// TwinCAT 3 PLC project PlcProj
// ProgramVersion: 3.1.4024.12
// libraries:
//   Tc2_BABasic, * (Beckhoff Automation GmbH)
//   Tc2_Drive, * (Beckhoff Automation GmbH)
//   Tc2_MC2, * (Beckhoff Automation GmbH)
//   Tc2_MC2_Drive, * (Beckhoff Automation GmbH)
//   Tc2_NcKinematicTransformation, * (Beckhoff Automation GmbH)
//   Tc2_PlcInterpolation, * (Beckhoff Automation GmbH)
//   Tc2_Standard, * (Beckhoff Automation GmbH)
//   Tc2_System, * (Beckhoff Automation GmbH)
//   Tc2_Utilities, * (Beckhoff Automation GmbH)
//   Tc3_McCoordinatedMotion, * (Beckhoff Automation GmbH)
//   Tc3_Module, * (Beckhoff Automation GmbH)
// project tree:
//   FBs/ FB_CalculateLinkageArm.TcPOU, FB_EnableAxes.TcPOU, FB_ResetCoordinateAxes.TcPOU
//   GVLs/ GVL.TcGVL
//   / PlcTask.TcTTO
//   POUs/ MAIN.TcPOU
// real-time tasks:
//   TASK PlcTask: cycle T#10ms, priority 20, ADS port 350
//   TASK Job Task: cycle default, priority 32
// motion (NC):
//   TASK NC-Task 1 SAF: cycle T#2ms, priority 4, ADS port 501
//   TASK NC-Task 1 SVB: cycle T#10ms, priority 8, ADS port 511
//   AXIS M1 (ACS) Degrees (id 1)
//     PositionAreaControl: Enable=false, Range=0
//     OtherSettings: AllowMotionCmdToSlave=true
//     encoder EncType=1
//     drive DrvType=5
//       Analog: TorqueSetpointScale=10, ScaleFactorActTorque=0.1
//       TimeComp: TaskDelayCycles=1
//     controller CtrType=1
//       CtrPara: PriorControlFactor=1
//         PosDiffControl: Enable=false, Range=0
//         Observer: BandWidth=20
//   AXIS M2 (ACS) Degrees (id 2)
//     PositionAreaControl: Enable=false, Range=0
//     OtherSettings: AllowMotionCmdToSlave=true
//     encoder EncType=1
//     drive DrvType=5
//       Analog: TorqueSetpointScale=10, ScaleFactorActTorque=0.1
//       TimeComp: TaskDelayCycles=1
//     controller CtrType=1
//       CtrPara: PriorControlFactor=1
//         PosDiffControl: Enable=false, Range=0
//         Observer: BandWidth=20
//   AXIS M3 (ACS) mm (id 3)
//     PositionAreaControl: Enable=false, Range=0
//     OtherSettings: AllowMotionCmdToSlave=true
//     encoder EncType=1
//     drive DrvType=5
//       Analog: TorqueSetpointScale=10, ScaleFactorActTorque=0.1
//       TimeComp: TaskDelayCycles=1
//     controller CtrType=1
//       CtrPara: PriorControlFactor=1
//         PosDiffControl: Enable=false, Range=0
//         Observer: BandWidth=20
//   AXIS M4 (ACS) Degrees (id 4)
//     PositionAreaControl: Enable=false, Range=0
//     OtherSettings: AllowMotionCmdToSlave=true
//     encoder EncType=1
//     drive DrvType=5
//       Analog: TorqueSetpointScale=10, ScaleFactorActTorque=0.1
//       TimeComp: TaskDelayCycles=1
//     controller CtrType=1
//       CtrPara: PriorControlFactor=1
//         PosDiffControl: Enable=false, Range=0
//         Observer: BandWidth=20
//   AXIS X (MCS) (id 5)
//     OtherSettings: AllowMotionCmdToSlave=true
//     encoder EncType=1
//     drive DrvType=5
//       Analog: TorqueSetpointScale=10, ScaleFactorActTorque=0.1
//       TimeComp: TaskDelayCycles=1
//     controller CtrType=1
//       CtrPara: PriorControlFactor=1
//         Observer: BandWidth=20
//   AXIS Y (MCS) (id 6)
//     OtherSettings: AllowMotionCmdToSlave=true
//     encoder EncType=1
//     drive DrvType=5
//       Analog: TorqueSetpointScale=10, ScaleFactorActTorque=0.1
//       TimeComp: TaskDelayCycles=1
//     controller CtrType=1
//       CtrPara: PriorControlFactor=1
//         Observer: BandWidth=20
//   AXIS Z (MCS) (id 7)
//     OtherSettings: AllowMotionCmdToSlave=true
//     encoder EncType=1
//     drive DrvType=5
//       Analog: TorqueSetpointScale=10, ScaleFactorActTorque=0.1
//       TimeComp: TaskDelayCycles=1
//     controller CtrType=1
//       CtrPara: PriorControlFactor=1
//         Observer: BandWidth=20
//   AXIS C (MCS) (id 8)
//     OtherSettings: AllowMotionCmdToSlave=true
//     encoder EncType=1
//     drive DrvType=5
//       Analog: TorqueSetpointScale=10, ScaleFactorActTorque=0.1
//       TimeComp: TaskDelayCycles=1
//     controller CtrType=1
//       CtrPara: PriorControlFactor=1
//         Observer: BandWidth=20
// variable links:
//   PlcProj/PlcProj Instance <-> NC-Task 1 SAF/Axes/C (MCS)
//     PlcTask Inputs/MAIN.io_C.NcToPlc <-> Outputs/ToPlc
//     PlcTask Outputs/MAIN.io_C.PlcToNc <-> Inputs/FromPlc
//   PlcProj/PlcProj Instance <-> NC-Task 1 SAF/Axes/M1 (ACS) Degrees
//     PlcTask Inputs/MAIN.io_M1.NcToPlc <-> Outputs/ToPlc
//     PlcTask Outputs/MAIN.io_M1.PlcToNc <-> Inputs/FromPlc
//   PlcProj/PlcProj Instance <-> NC-Task 1 SAF/Axes/M2 (ACS) Degrees
//     PlcTask Inputs/MAIN.io_M2.NcToPlc <-> Outputs/ToPlc
//     PlcTask Outputs/MAIN.io_M2.PlcToNc <-> Inputs/FromPlc
//   PlcProj/PlcProj Instance <-> NC-Task 1 SAF/Axes/M3 (ACS) mm
//     PlcTask Inputs/MAIN.io_M3.NcToPlc <-> Outputs/ToPlc
//     PlcTask Outputs/MAIN.io_M3.PlcToNc <-> Inputs/FromPlc
//   PlcProj/PlcProj Instance <-> NC-Task 1 SAF/Axes/M4 (ACS) Degrees
//     PlcTask Inputs/MAIN.io_M4.NcToPlc <-> Outputs/ToPlc
//     PlcTask Outputs/MAIN.io_M4.PlcToNc <-> Inputs/FromPlc
//   PlcProj/PlcProj Instance <-> NC-Task 1 SAF/Axes/X (MCS)
//     PlcTask Inputs/MAIN.io_X.NcToPlc <-> Outputs/ToPlc
//     PlcTask Outputs/MAIN.io_X.PlcToNc <-> Inputs/FromPlc
//   PlcProj/PlcProj Instance <-> NC-Task 1 SAF/Axes/Y (MCS)
//     PlcTask Inputs/MAIN.io_Y.NcToPlc <-> Outputs/ToPlc
//     PlcTask Outputs/MAIN.io_Y.PlcToNc <-> Inputs/FromPlc
//   PlcProj/PlcProj Instance <-> NC-Task 1 SAF/Axes/Z (MCS)
//     PlcTask Inputs/MAIN.io_Z.NcToPlc <-> Outputs/ToPlc
//     PlcTask Outputs/MAIN.io_Z.PlcToNc <-> Inputs/FromPlc
//   PlcProj/PlcProj Instance <-> NC-Task 1 SAF/Kinematics Channel
//     PlcTask Inputs/MAIN.in_stKinToPlc <-> Outputs/ToPlc
//     PlcTask Outputs/MAIN.out_stPlcToKin <-> Inputs/FromPlc
//   PlcProj/PlcProj Instance <-> NC-Task 1 SAF/Objects/Motion Group
//     PlcTask Inputs/GVL.stGroupRef.NcToPlc <-> Group Outputs/ToPLC
//     PlcTask Outputs/GVL.stGroupRef.PlcToNc <-> Group Inputs/FromPLC

CONFIGURATION PlcProj
    RESOURCE PLC ON TwinCAT3
        TASK PlcTask(INTERVAL := T#10ms, PRIORITY := 20);
        PROGRAM MAIN WITH PlcTask : MAIN;
    END_RESOURCE
END_CONFIGURATION

// ---- GVLs/GVL.TcGVL
{attribute 'qualified_only'}
VAR_GLOBAL
	
	stGroupRef : AXES_GROUP_REF;
	{attribute 'TcInitSymbol'}  oidConveyorBelt : MC_COORD_REF;

	
END_VAR

// ---- POUs/MAIN.TcPOU
PROGRAM MAIN
VAR
	
	inner_arm : FB_CalculateLinkageArm;
	outer_arm : FB_CalculateLinkageArm;
	
	io_X:	AXIS_REF;
	io_Y:	AXIS_REF;
	io_Z:	AXIS_REF;
	io_C:	AXIS_REF;	
	io_M1:	AXIS_REF;
	io_M2:	AXIS_REF;
	io_M3:	AXIS_REF;
	io_M4:	AXIS_REF;	

	fbAddAxisXtoGrp : MC_AddAxisToGroup;
	fbAddAxisYtoGrp : MC_AddAxisToGroup;
	fbAddAxisZtoGrp : MC_AddAxisToGroup;	
	fbAddAxisCtoGrp : MC_AddAxisToGroup;	
	
//	Kinematic Functions / Structures / Vars
	bkinConfigGrp				: BOOL;
	bkinCartesianMode			: BOOL := TRUE; //When bCartesianMode is TRUE, movement in the MCS (Cartesian) axes will be transformed into the ACS (Joint) axes. The ACS axes cannot be moved directly.
	bkinResetGrp					: BOOL;
	in_stKinToPlc	AT %I*		: NcToPlc_NciChannel_Ref;
	out_stPlcToKin	AT %Q*		: PLCTONC_NCICHANNEL_REF;
	stAxesConfig				: ST_KinAxes;
	fbCalcTrafo					: FB_KinCalcTrafo;
	metaIn						: U_KinMetaInfo;
	metaOut						: U_KinMetaInfo;
	fbKinConfigGrp				: FB_KinConfigGroup;  //Configures ACS and MCS axes to the kinematic transformation group
	fbKinResetGrp				: FB_KinResetGroup;  //Resets the kinematic transformation group
	oidTrafo		AT %I*		: OTCID;
	kinStatus 					: E_KinStatus;
	
	bDeltaKinEnable : BOOL;
	bDeltaKinReady : BOOL;
	bDeltaKinActive : BOOL;
	bDeltaKinInactive : BOOL;
	nDeltaKinState : INT;
	
	bKinGrpEnable : BOOL;
	bKinGrpReady : BOOL;
	bKinGrpError : BOOL;
	bKinGrpReset : BOOL;
	bNciEnable : BOOL;
	bKinResetDone : BOOL;
	bNciReadytToEnable : BOOL;
	bEnableAxes : BOOL;
	bAllAxesReady : BOOL;
	fbKinDelay : TON;
	fbEnableAxes : FB_EnableAxes;
	bAxisFault : BOOL;
	fbResetCoordinateAxes : FB_ResetCoordinateAxes;
	fbJogX : MC_Jog;
	fbJogY : MC_Jog;
	fbJogZ : MC_Jog;
	fbMoveX : MC_MoveRelative;
	bMoveX : BOOL;
	nDistanceX : INT;
	nDistanceY : INT;
	nDistanceZ : INT;
	bMoveY : BOOL;
	bMoveZ : BOOL;
	fbMoveY : MC_MoveRelative;
	fbMoveZ : MC_MoveRelative;
	bAxesNotMoving : BOOL;
	bJogXpos : BOOL;
	bJogXneg : BOOL;
	nMoveState	: WORD;
	
	bMotionGrpEnable : BOOL;	// Enable the Motion Group
	bMotionGrpBuild : BOOL;		// Add Axes To Motion Group
	bMotionGrpStop : BOOL;
	bMotionGrpStart : BOOL;
	bMotionGrpPrep : BOOL;
	bMotionGrpOvr : BOOL;
	
	fbMgSetOverride : MC_GroupSetOverride;
	fbMgEnable : MC_GroupEnable;
	fbMoveLinPrep : MC_MoveLinearAbsolutePreparation;
	fbMoveCircPrep : MC_MoveCircularAbsolutePreparation;
	fbMgMovePath : MC_MovePath;
	fbMgStop 	: MC_GroupStop;
	fbMgReadStatus : MC_GroupReadStatus;
	
	// hmi
	
	nDisplayZ : LREAL;
	nPkgZ   : LREAL;
	nScaleZ : LREAL;
	nDisplayX : LREAL;
	nDisplayY : LREAL;
	
	
	// copied from sample proj
	
	buffer					: ARRAY[1..4096] OF BYTE;
	path					: MC_PATH_DATA_REF(ADR(buffer), SIZEOF(buffer));
	
	aTargetPos				: ARRAY[1..4] OF MC_LREAL;
	aTransitionParam		: ARRAY[1..2] OF MC_LREAL;
	aAuxPoint                               : ARRAY[1..3] OF MC_LREAL;
	fVelFactor				: LREAL := 1.0;
	bMovePrepError : BOOL;
	bBarPicked : BOOL;
	bAddNewBar : BOOL;
	fbAddNewBar : TON;
	bBarPlaced : BOOL;
	nBarDisplayX : LREAL;
	nBarDisplayY : LREAL;
	nBarDisplayZ : LREAL;
	bNewPath	: BOOL;
	bBarInPlace  : BOOL;
	nTestBarX : LREAL;
	nTestBarY : LREAL;
	nTestBarZ : LREAL;
		nScaledBarX : LREAL;
	nScaledBarY : LREAL;
	nScaledBarZ : LREAL;
	
	
	fbTrackConveyor : MC_TrackConveyorBelt;
	MasterRefPos : MC_LREAL;
	InitialObjectPos : ARRAY [1..4] OF MC_LREAL;
	bStartTracking : BOOL;
	fbStartConveyor : MC_MoveVelocity;
	fbStopConveyor : MC_Stop;
	bStartConveyor : BOOL;
	bStopGroup : BOOL;
	lrYpos: MC_LREAL;
	fbSetM1Pos : MC_SetPosition;
	fbSetM2Pos : MC_SetPosition;
	fbSetM4Pos : MC_SetPosition;
	bSetPos : BOOL;
	
	nTrackX: LREAL;
END_VAR


// action calls
	Main.cartesian_ops();
	Main.kinematic_ops();
	Main.motion_group();

// calculations for hmi display of the scara linkages
	inner_arm(
		x0:= 375, 
		y0:= 375, 
		theta:= io_M1.NcToPlc.ActPos, 
		L:= 190, 
		x1=> , 
		y1=> );
	
	outer_arm(
		x0:= inner_arm.x1, 
		y0:= inner_arm.y1, 
		theta:= io_M2.NcToPlc.ActPos, 
		L:= 190, 
		x1=> , 
		y1=> );

// Axis Ref Read Status
	io_X.ReadStatus();
	io_Y.ReadStatus();
	io_Z.ReadStatus();
	io_C.ReadStatus();	
	io_M1.ReadStatus();
	io_M2.ReadStatus();
	io_M3.ReadStatus();
	io_M4.ReadStatus();	

// check for motor movement
	bAxesNotMoving := io_M1.Status.NotMoving AND io_M2.Status.NotMoving AND io_M3.Status.NotMoving AND io_M4.Status.NotMoving;
	
// read axes id's from cylic interface so they can mapped later to the kinematic group
	stAxesConfig.nAxisIdsAcs[1]	:= io_M1.NcToPlc.AxisId;
	stAxesConfig.nAxisIdsAcs[2]	:= io_M2.NcToPlc.AxisId;
	stAxesConfig.nAxisIdsAcs[3]	:= io_M3.NcToPlc.AxisId;
	stAxesConfig.nAxisIdsAcs[4]	:= io_M4.NcToPlc.AxisId;	
	stAxesConfig.nAxisIdsMcs[1]	:= io_X.NcToPlc.AxisId;
	stAxesConfig.nAxisIdsMcs[2]	:= io_Y.NcToPlc.AxisId;
	stAxesConfig.nAxisIdsMcs[3]	:= io_Z.NcToPlc.AxisId;
	stAxesConfig.nAxisIdsMcs[4]	:= io_C.NcToPlc.AxisId;	
	

	fbMgMovePath(
		AxesGroup:= GVL.stGroupRef , 
		PathData:= path , 
		Execute:= bMotionGrpStart
	);
	
	fbMgStop(
		AxesGroup := GVL.stGroupRef,
		Execute	:= bStopGroup
		);
	
			
CASE nMoveState OF
	
1:	//	init

		nMoveState	:= 4;
		
4:	// set up path data for the pick position

		Main.prep_pick_path();
		//Main.prep_start_path();
		
		IF path.FilledRows > 0 THEN
			nMoveState	:= 5;
		END_IF
		
5:	// move to the pick psoition

		bMotionGrpStart := TRUE;

		IF fbMgMovePath.Done THEN
			bMotionGrpStart := FALSE;
			nMoveState := 100;
		END_IF

10:	// set up path data for the place position

		Main.prep_place_path();
		//Main.prep_finish_path();
		
		IF path.FilledRows > 0 THEN
			nMoveState	:= 15;
		END_IF
		
15:	// move to the place position

		bMotionGrpStart := TRUE;

		IF fbMgMovePath.Done THEN
			bMotionGrpStart := FALSE;
			nMoveState := 1;
		END_IF

100: // stopping...

		bStopGroup := TRUE;
		
		IF fbMgStop.Done THEN
			bStopGroup := FALSE;
			nMoveState	:= 10;
		END_IF		

END_CASE

ACTION cartesian_ops:
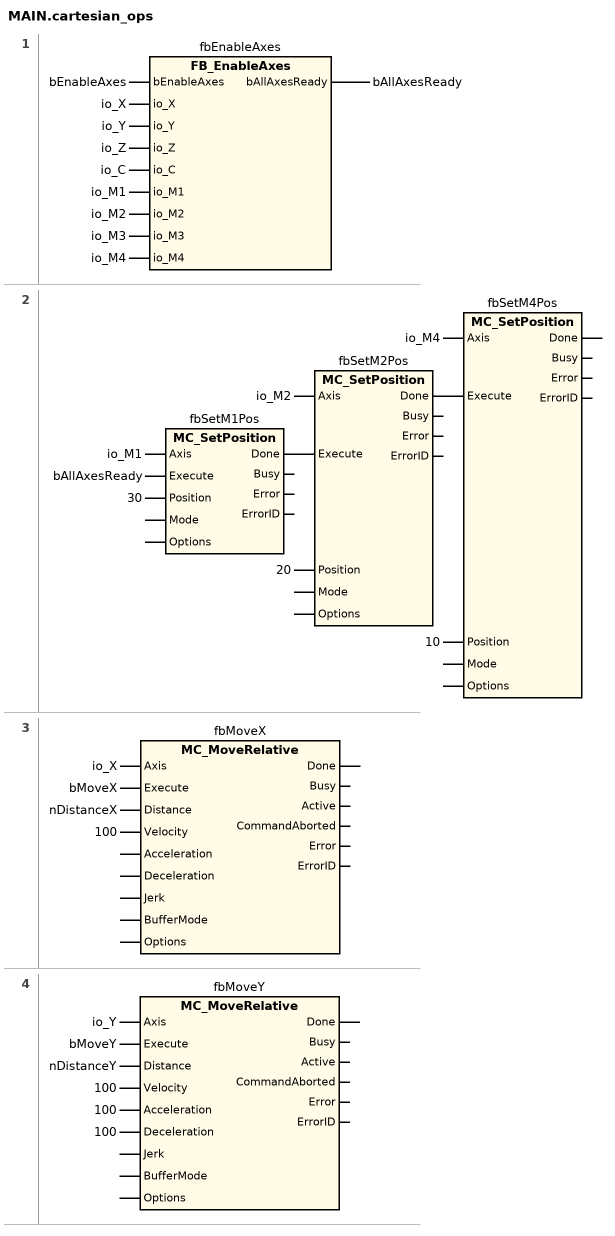
// NETWORK 1
fbEnableAxes(
    bEnableAxes := bEnableAxes,
    io_X := io_X,
    io_Y := io_Y,
    io_Z := io_Z,
    io_C := io_C,
    io_M1 := io_M1,
    io_M2 := io_M2,
    io_M3 := io_M3,
    io_M4 := io_M4); // FB_EnableAxes
bAllAxesReady := fbEnableAxes.bAllAxesReady;

// NETWORK 2
fbSetM1Pos(Axis := io_M1, Execute := bAllAxesReady, Position := 30); // MC_SetPosition
fbSetM2Pos(Axis := io_M2, Execute := fbSetM1Pos.Done, Position := 20); // MC_SetPosition
fbSetM4Pos(Axis := io_M4, Execute := fbSetM2Pos.Done, Position := 10); // MC_SetPosition

// NETWORK 3
fbMoveX(Axis := io_X, Execute := bMoveX, Distance := nDistanceX, Velocity := 100); // MC_MoveRelative

// NETWORK 4
fbMoveY(
    Axis := io_Y,
    Execute := bMoveY,
    Distance := nDistanceY,
    Velocity := 100,
    Acceleration := 100,
    Deceleration := 100); // MC_MoveRelative

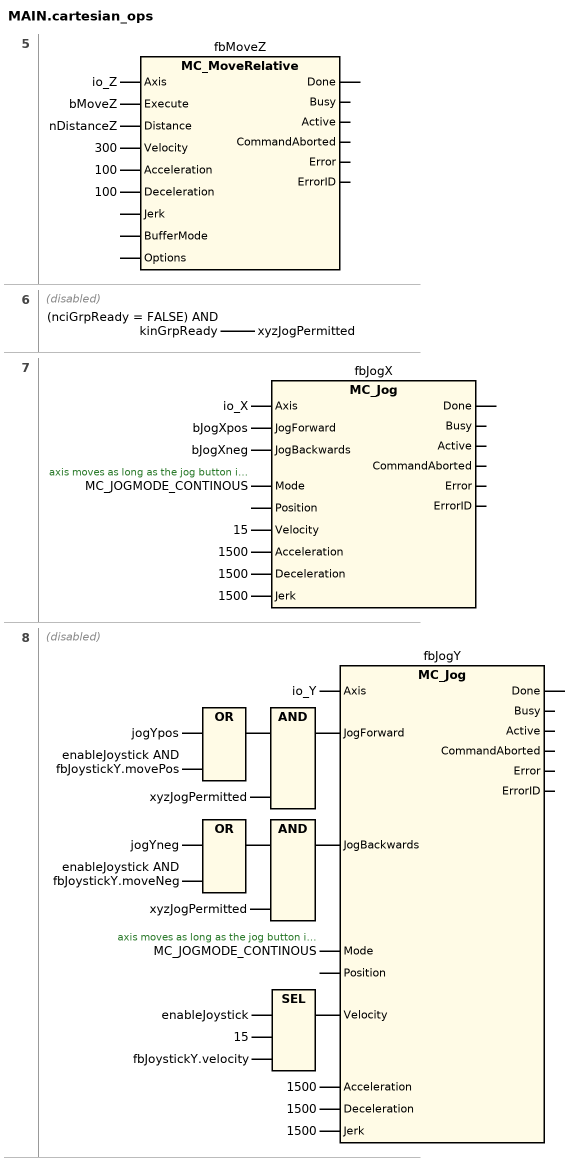
// NETWORK 5
fbMoveZ(
    Axis := io_Z,
    Execute := bMoveZ,
    Distance := nDistanceZ,
    Velocity := 300,
    Acceleration := 100,
    Deceleration := 100); // MC_MoveRelative

// NETWORK 6 (disabled)
// xyzJogPermitted := (nciGrpReady = FALSE) AND kinGrpReady;

// NETWORK 7
//   MC_JOGMODE_CONTINOUS: axis moves as long as the jog button is pressed using parameterized dynamics
fbJogX(
    Axis := io_X,
    JogForward := bJogXpos,
    JogBackwards := bJogXneg,
    Mode := MC_JOGMODE_CONTINOUS,
    Velocity := 15,
    Acceleration := 1500,
    Deceleration := 1500,
    Jerk := 1500); // MC_Jog

// NETWORK 8 (disabled)
//   MC_JOGMODE_CONTINOUS: axis moves as long as the jog button is pressed using parameterized dynamics
// fbJogY(
//     Axis := io_Y,
//     JogForward := (jogYpos OR (enableJoystick AND fbJoystickY.movePos)) AND xyzJogPermitted,
//     JogBackwards := (jogYneg OR (enableJoystick AND fbJoystickY.moveNeg)) AND xyzJogPermitted,
//     Mode := MC_JOGMODE_CONTINOUS,
//     Velocity := SEL(enableJoystick, 15, fbJoystickY.velocity),
//     Acceleration := 1500,
//     Deceleration := 1500,
//     Jerk := 1500); // MC_Jog

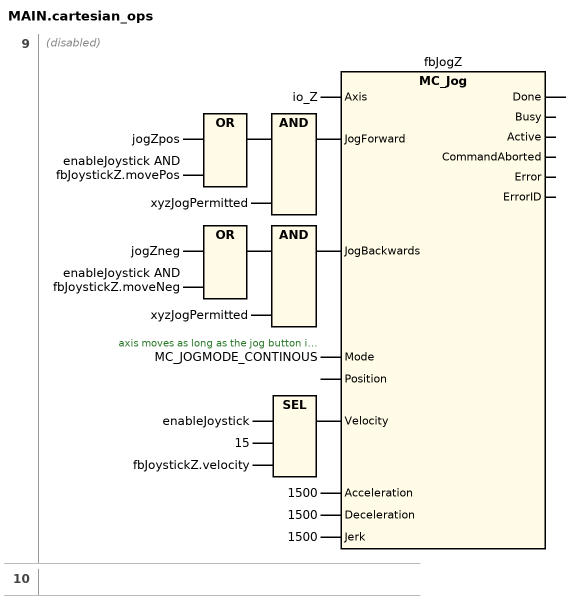
// NETWORK 9 (disabled)
//   MC_JOGMODE_CONTINOUS: axis moves as long as the jog button is pressed using parameterized dynamics
// fbJogZ(
//     Axis := io_Z,
//     JogForward := (jogZpos OR (enableJoystick AND fbJoystickZ.movePos)) AND xyzJogPermitted,
//     JogBackwards := (jogZneg OR (enableJoystick AND fbJoystickZ.moveNeg)) AND xyzJogPermitted,
//     Mode := MC_JOGMODE_CONTINOUS,
//     Velocity := SEL(enableJoystick, 15, fbJoystickZ.velocity),
//     Acceleration := 1500,
//     Deceleration := 1500,
//     Jerk := 1500); // MC_Jog

// NETWORK 10
END_ACTION

ACTION kinematic_ops:
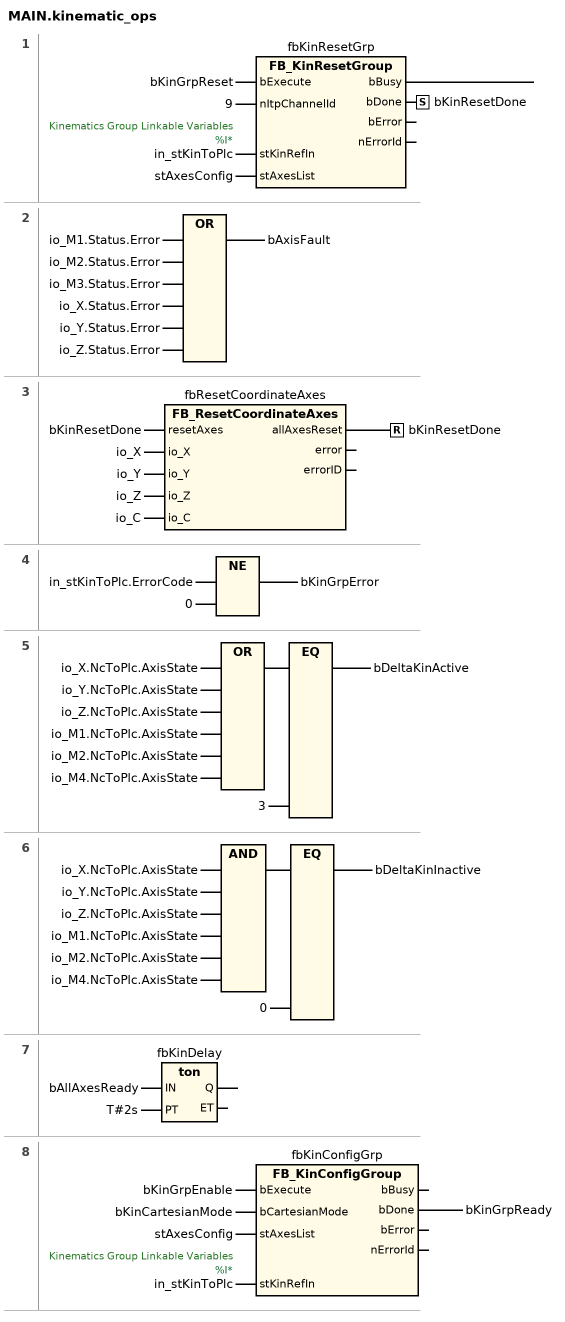
// NETWORK 1
//   fbKinResetGrp: Resets the kinematic transformation group
//   in_stKinToPlc: Kinematics Group Linkable Variables | AT %I*
fbKinResetGrp(
    bExecute := bKinGrpReset,
    nItpChannelId := 9,
    stKinRefIn := in_stKinToPlc,
    stAxesList := stAxesConfig); // FB_KinResetGroup
bKinResetDone S= fbKinResetGrp.bDone;

// NETWORK 2
bAxisFault := io_M1.Status.Error OR io_M2.Status.Error OR io_M3.Status.Error OR io_X.Status.Error OR io_Y.Status.Error OR io_Z.Status.Error;

// NETWORK 3
fbResetCoordinateAxes(resetAxes := bKinResetDone, io_X := io_X, io_Y := io_Y, io_Z := io_Z, io_C := io_C); // FB_ResetCoordinateAxes
bKinResetDone R= fbResetCoordinateAxes.allAxesReset;

// NETWORK 4
bKinGrpError := in_stKinToPlc.ErrorCode <> 0;

// NETWORK 5
bDeltaKinActive := (io_X.NcToPlc.AxisState OR io_Y.NcToPlc.AxisState OR io_Z.NcToPlc.AxisState OR io_M1.NcToPlc.AxisState OR io_M2.NcToPlc.AxisState OR io_M4.NcToPlc.AxisState) = 3;

// NETWORK 6
bDeltaKinInactive := (io_X.NcToPlc.AxisState AND io_Y.NcToPlc.AxisState AND io_Z.NcToPlc.AxisState AND io_M1.NcToPlc.AxisState AND io_M2.NcToPlc.AxisState AND io_M4.NcToPlc.AxisState) = 0;

// NETWORK 7
fbKinDelay(IN := bAllAxesReady, PT := T#2s); // ton

// NETWORK 8
//   fbKinConfigGrp: Configures ACS and MCS axes to the kinematic transformation group
//   in_stKinToPlc: Kinematics Group Linkable Variables | AT %I*
fbKinConfigGrp(
    bExecute := bKinGrpEnable,
    bCartesianMode := bKinCartesianMode,
    stAxesList := stAxesConfig,
    stKinRefIn := in_stKinToPlc); // FB_KinConfigGroup
bKinGrpReady := fbKinConfigGrp.bDone;

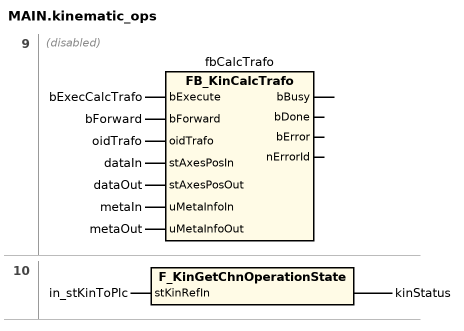
// NETWORK 9 (disabled)
// fbCalcTrafo(
//     bExecute := bExecCalcTrafo,
//     bForward := bForward,
//     oidTrafo := oidTrafo,
//     stAxesPosIn := dataIn,
//     stAxesPosOut := dataOut,
//     uMetaInfoIn := metaIn,
//     uMetaInfoOut := metaOut); // FB_KinCalcTrafo

// NETWORK 10
kinStatus := F_KinGetChnOperationState(stKinRefIn := in_stKinToPlc);
END_ACTION

ACTION kinematic_sm:

(*
		setStartPos[5](Axis:= io_X, 
			Execute:= setZeroPosition,
			Position:= 0);
		setStartPos[6](Axis:= io_Y,
			Execute:= setZeroPosition, 
			Position:= 0);
		setStartPos[7](Axis:= io_Z, 
			Execute:= setZeroPosition,
			Position:= 0);
*)

CASE nDeltaKinState OF 

0: 	nDeltaKinState := 2;

		
2:			// RESET ALL NCI VARIABLES
		//nciRunProgram := FALSE;
		//nciBuildTable := FALSE;
		//nciResetTable := TRUE;
		//nciResetProgram := TRUE;
		nDeltaKinState := 3;
		
3:
		//nciResetProgram := FALSE;
		//nciResetTable := FALSE;
		nDeltaKinState := 4;
		
4:			// RESET ALL KINEMATIC VARIABLES
		IF bKinGrpError THEN
				bKinGrpReset := TRUE;
				nDeltaKinState :=5;
		ELSIF bKinGrpError = FALSE THEN
				nDeltaKinState := 104;
		END_IF
				
5:
		bKinGrpReset := FALSE;
		nDeltaKinState := 4;
		
104:		// RESET ALL KINEMATIC VARIABLES
		IF bAxisFault THEN
				bKinGrpReset := TRUE;
				nDeltaKinState :=105;
		ELSIF bAxisFault = FALSE THEN
				nDeltaKinState := 6;
		END_IF
				
105:
		bKinGrpReset := FALSE;
		nDeltaKinState := 104;

6: 		// IF IN START POSITION - ENABLE AXES
		nDeltaKinState := 7;

7:			// ALL AXES ARE POWERED
		IF bAllAxesReady AND bAxesNotMoving THEN
				nDeltaKinState := 8;
		END_IF
		
8:			// ENABLE KINEMATIC GROUP FUNCTION
		nDeltaKinState := 9;
			
9: 		// DELAY TO ALLOW KINEMATIC GROUP TIME TO PROCESS REQUEST
		IF fbKinDelay.Q AND bKinGrpReady AND bAxesNotMoving THEN
				nDeltaKinState := 10;
		END_IF
	(*	
10:		// ENABLE NCI BUILD GROUP

		nDeltaKinState := 11;

11: 	// WAIT FOR BUILD GROUP DONE AND ADDITIONAL DELAY BEFORE STARTING BUILD TABLE
		IF kinGrpReady  AND  tNciDelay.Q THEN 
				nciBuildTable := TRUE;
				nDeltaKinState := 12;
		ELSIF kinGrpReady = FALSE THEN
				nDeltaKinState := 50;
		END_IF

12: 	// WAIT FOR ROWS TO BE FILLED

		IF fbNciFeedTablePrep.nFilledRows > 0 THEN
				nciBuildTable := FALSE;
				nDeltaKinState:= 13;
		END_IF

13:	// RUN COMMAND WILL START THE NCI FEED TABLE PROGRAM
		IF nciRunCmd  THEN
				nciRunProgram := TRUE; 	
				nDeltaKinState :=14;
		ELSIF nciEnable = FALSE THEN
				nDeltaKinState := 0;
		END_IF
		
14:	
		IF nciFeedingDone THEN
				nciRunProgram := FALSE;
				nDeltaKinState := 15;
		ELSIF nciEnable = FALSE THEN
				nDeltaKinState := 0;
		END_IF

15:	// REACHED END OF FEED TABLE PROGRAM
		IF fbNciTable.bChannelDone THEN
				nDeltaKinState	:= 16;
		ELSIF nciEnable = FALSE THEN
				nDeltaKinState := 0;
		END_IF
		
16:	// IF RUN IS STILL ACTIVE, LOOP BACK THROUGH THE FEED TABLE PROGRAM

		nDeltaKinState := 13;


50: // DECOUPLE KINEMATIC GROUP FROM AXES
		kinCartesianMode := FALSE;
		kinGrpEnable := TRUE;
		
		IF kinStatus = KinStatus_Empty THEN
				kinCartesianMode := TRUE;
				kinGrpEnable := FALSE;
				nDeltaKinState := 4;
		END_IF
	*)			
END_CASE
END_ACTION

ACTION motion_group:
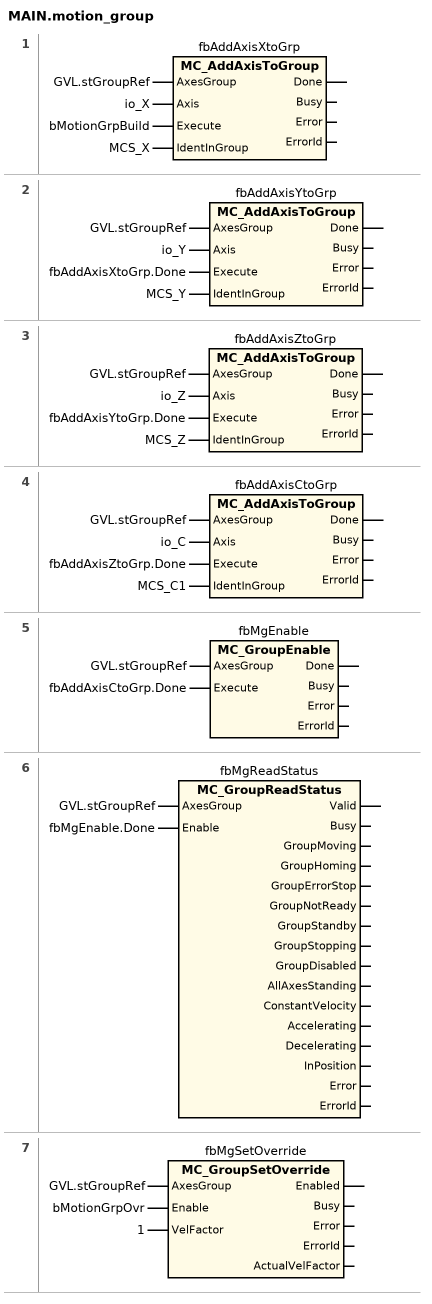
// NETWORK 1
fbAddAxisXtoGrp(AxesGroup := GVL.stGroupRef, Axis := io_X, Execute := bMotionGrpBuild, IdentInGroup := MCS_X); // MC_AddAxisToGroup

// NETWORK 2
fbAddAxisYtoGrp(
    AxesGroup := GVL.stGroupRef,
    Axis := io_Y,
    Execute := fbAddAxisXtoGrp.Done,
    IdentInGroup := MCS_Y); // MC_AddAxisToGroup

// NETWORK 3
fbAddAxisZtoGrp(
    AxesGroup := GVL.stGroupRef,
    Axis := io_Z,
    Execute := fbAddAxisYtoGrp.Done,
    IdentInGroup := MCS_Z); // MC_AddAxisToGroup

// NETWORK 4
fbAddAxisCtoGrp(
    AxesGroup := GVL.stGroupRef,
    Axis := io_C,
    Execute := fbAddAxisZtoGrp.Done,
    IdentInGroup := MCS_C1); // MC_AddAxisToGroup

// NETWORK 5
fbMgEnable(AxesGroup := GVL.stGroupRef, Execute := fbAddAxisCtoGrp.Done); // MC_GroupEnable

// NETWORK 6
fbMgReadStatus(AxesGroup := GVL.stGroupRef, Enable := fbMgEnable.Done); // MC_GroupReadStatus

// NETWORK 7
fbMgSetOverride(AxesGroup := GVL.stGroupRef, Enable := bMotionGrpOvr, VelFactor := 1); // MC_GroupSetOverride
END_ACTION

ACTION prep_finish_path:

path.ClearPath();  //Clear nodes that were in path


// XYZ POSITIONS LIMITS
// X : -760 to +760
// Y : -760 to +760
// Z : 



fbMoveCircPrep.EndPoint                 	:= ADR(aTargetPos);
fbMoveCircPrep.EndPointCount            	:= 4;
fbMoveCircPrep.AuxPoint                 	:= ADR(aTransitionParam);
fbMoveCircPrep.AuxPointCount            	:= 3;
fbMoveCircPrep.CircMode                 	:= mcCircModeCenter;
fbMoveCircPrep.TransitionParameter      	:= ADR(aTransitionParam);
fbMoveCircPrep.TransitionParameterCount 	:= 2;
fbMoveCircPrep.BufferMode               	:= mcBlendingPrevious;
fbMoveCircPrep.TransitionMode           	:= mcTransModeNone;
	
fbMoveLinPrep.Position						:= ADR(aTargetPos); //pointer to position array
fbMoveLinPrep.PositionCount 				:= 4; //number of axes in group
fbMoveLinPrep.TransitionParameter			:= ADR (aTransitionParam); //pointer to transition parameter array
fbMoveLinPrep.TransitionParameterCount		:= 2; //number of transition parameters, has to be set always 2
fbMoveLinPrep.BufferMode					:= mcBlendingPrevious;
fbMoveLinPrep.TransitionMode				:= mcTransModeCornerDistanceAdvanced;

//Set dynamics to default values of the axes
fbMoveLinPrep.Acceleration					:= MC_DEFAULT;
fbMoveLinPrep.Deceleration					:= MC_DEFAULT;
fbMoveLinPrep.Jerk							:= MC_DEFAULT;

bMovePrepError := bMovePrepError OR fbMoveLinPrep.Error;



  	aTargetPos[1]                           := 625;
    aTargetPos[2]                           := 10;
    aTargetPos[3]                           := 0;
    aTransitionParam[1]                     := 0;
    aTransitionParam[2]                     := 0;
    fbMoveLinPrep(PathData:= path, Velocity:= 100, InvokeId:= 10);

    aTargetPos[1]                           := -400;
    aTargetPos[2]                           := -300;
    aTargetPos[3]                           := 0;
    aAuxPoint[1]                            := -357.5;
    aAuxPoint[2]                            := -257.5;
    aAuxPoint[3]                            := 0;
    aTransitionParam[1]                     := 0;
    aTransitionParam[2]                     := 0;
    fbMoveCircPrep(PathData:= path, PathChoice:= mcCircPathchoiceClockwise, Velocity:= 100, InvokeId:= 20);
END_ACTION

ACTION prep_pick_path:
path.ClearPath();  //Clear nodes that were in path


// XYZ POSITIONS LIMITS
// X : -760 to +760
// Y : -760 to +760
// Z : 

//1st node
aTargetPos[1]				:=634;		// X Position
aTargetPos[2]				:= 10;		// Y Position
aTargetPos[3]				:= 0;	// Z Position
aTargetPos[4]				:= 0;	// C Position
aTransitionParam[1]			:= 0; //blending distance on previous segment, no influence here
aTransitionParam[2]			:= 0; //blending distance on this segment, no influence here
fbMoveLinPrep(PathData:= path , Velocity:= 200, InvokeId:= 10);
bMovePrepError := bMovePrepError OR fbMoveLinPrep.Error;

fbMoveLinPrep.Position						:= ADR(aTargetPos); //pointer to position array
fbMoveLinPrep.PositionCount 				:= 4; //number of axes in group
fbMoveLinPrep.TransitionParameter			:= ADR (aTransitionParam); //pointer to transition parameter array
fbMoveLinPrep.TransitionParameterCount		:= 2; //number of transition parameters, has to be set always 2
fbMoveLinPrep.BufferMode					:= mcBlendingPrevious;
fbMoveLinPrep.TransitionMode				:= mcTransModeCornerDistanceAdvanced;
//Set dynamics to default values of the axes
fbMoveLinPrep.Acceleration					:= MC_DEFAULT;
fbMoveLinPrep.Deceleration					:= MC_DEFAULT;
fbMoveLinPrep.Jerk							:= MC_DEFAULT;
END_ACTION

ACTION prep_place_path:
path.ClearPath();  //Clear nodes that were in path

// XYZ POSITIONS LIMITS
// X : -550 to +550
// Y : -550 to +550
// Z : -750 to -950

fbMoveLinPrep.Position						:= ADR(aTargetPos); //pointer to position array
fbMoveLinPrep.PositionCount 				:= 4; //number of axes in group
fbMoveLinPrep.TransitionParameter			:= ADR (aTransitionParam); //pointer to transition parameter array
fbMoveLinPrep.TransitionParameterCount		:= 2; //number of transition parameters, has to be set always 2
fbMoveLinPrep.BufferMode					:= mcBlendingPrevious;
fbMoveLinPrep.TransitionMode				:= mcTransModeCornerDistanceAdvanced;
//Set dynamics to default values of the axes
fbMoveLinPrep.Acceleration					:= MC_DEFAULT;
fbMoveLinPrep.Deceleration					:= MC_DEFAULT;
fbMoveLinPrep.Jerk							:= MC_DEFAULT;
(*
//1st node
aTargetPos[1]				:= -225;		// X Position
aTargetPos[2]				:= 225;		// Y Position
aTargetPos[3]				:= -900;	// Z Position
aTransitionParam[1]			:= 0; //blending distance on previous segment, no influence here
aTransitionParam[2]			:= 0; //blending distance on this segment, no influence here
fbMoveLinPrep(PathData:= path , Velocity:= 2100, InvokeId:= 10);
bMovePrepError := bMovePrepError OR fbMoveLinPrep.Error;

aTargetPos[1]				:= 225;
aTargetPos[2]				:= -225;
aTargetPos[3]				:= -750;
aTransitionParam[1]			:= 50; //blending distance on previous segment (InvokeId=10), defines when to leave line
aTransitionParam[2]			:= 50; //blending distance on this segment, defines latest positionn to be back  on line of InovkeId=20 
fbMoveLinPrep(PathData:= path , Velocity:= 2100, InvokeId:= 20); 
bMovePrepError := bMovePrepError OR fbMoveLinPrep.Error;

aTargetPos[1]				:= 225;
aTargetPos[2]				:= 225;
aTargetPos[3]				:= -950;
aTransitionParam[1]			:= 50; 
aTransitionParam[2]			:= 50;
fbMoveLinPrep(PathData:= path , Velocity:= 2100, InvokeId:= 30);
bMovePrepError := bMovePrepError OR fbMoveLinPrep.Error;

aTargetPos[1]				:= -225;
aTargetPos[2]				:= -225;
aTargetPos[3]				:= -750;
aTransitionParam[1]			:= 50; //blending distance on previous segment, no influence here
aTransitionParam[2]			:= 50; //blending distance on this segment, no influence here
fbMoveLinPrep(PathData:= path , Velocity:= 2100, InvokeId:= 40);
bMovePrepError := bMovePrepError OR fbMoveLinPrep.Error;
*)
aTargetPos[1]				:= -400;
aTargetPos[2]				:= -300;
aTargetPos[3]				:= 0;
aTargetPos[4]				:= 0;
aTransitionParam[1]			:= 50; 
aTransitionParam[2]			:= 50;
fbMoveLinPrep(PathData:= path , Velocity:= 150, InvokeId:= 50);
bMovePrepError := bMovePrepError OR fbMoveLinPrep.Error;
END_ACTION

ACTION prep_start_path:

path.ClearPath();  //Clear nodes that were in path


// XYZ POSITIONS LIMITS
// X : -760 to +760
// Y : -760 to +760
// Z : 



fbMoveCircPrep.EndPoint                 	:= ADR(aTargetPos);
fbMoveCircPrep.EndPointCount            	:= 4;
fbMoveCircPrep.AuxPoint                 	:= ADR(aTransitionParam);
fbMoveCircPrep.AuxPointCount            	:= 3;
fbMoveCircPrep.CircMode                 	:= mcCircModeCenter;
fbMoveCircPrep.TransitionParameter      	:= ADR(aTransitionParam);
fbMoveCircPrep.TransitionParameterCount 	:= 2;
fbMoveCircPrep.BufferMode               	:= mcBlendingPrevious;
fbMoveCircPrep.TransitionMode           	:= mcTransModeNone;
	
fbMoveLinPrep.Position						:= ADR(aTargetPos); //pointer to position array
fbMoveLinPrep.PositionCount 				:= 4; //number of axes in group
fbMoveLinPrep.TransitionParameter			:= ADR (aTransitionParam); //pointer to transition parameter array
fbMoveLinPrep.TransitionParameterCount		:= 2; //number of transition parameters, has to be set always 2
fbMoveLinPrep.BufferMode					:= mcBlendingPrevious;
fbMoveLinPrep.TransitionMode				:= mcTransModeCornerDistanceAdvanced;

//Set dynamics to default values of the axes
fbMoveLinPrep.Acceleration					:= MC_DEFAULT;
fbMoveLinPrep.Deceleration					:= MC_DEFAULT;
fbMoveLinPrep.Jerk							:= MC_DEFAULT;

bMovePrepError := bMovePrepError OR fbMoveLinPrep.Error;



  	aTargetPos[1]                           := -350;
    aTargetPos[2]                           := -300;
    aTargetPos[3]                           := 0;
    aTransitionParam[1]                     := 0;
    aTransitionParam[2]                     := 0;
    fbMoveLinPrep(PathData:= path, Velocity:= 100, InvokeId:= 10);

    aTargetPos[1]                           := 625;
    aTargetPos[2]                           := -10;
    aTargetPos[3]                           := 0;
    aAuxPoint[1]                            := 282.5;
    aAuxPoint[2]                            := -642.5;
    aAuxPoint[3]                            := 0;
    aTransitionParam[1]                     := 0;
    aTransitionParam[2]                     := 0;
    fbMoveCircPrep(PathData:= path, PathChoice:= mcCircPathChoiceCounterClockwise, Velocity:= 100, InvokeId:= 20);
END_ACTION

END_PROGRAM

// ---- FBs/FB_CalculateLinkageArm.TcPOU
FUNCTION_BLOCK FB_CalculateLinkageArm
VAR_INPUT
		x0 : REAL; 			(* Origin x-coordinate *)
        y0 : REAL; 			(* Origin y-coordinate *)
        theta : LREAL ;		(* Angle in degrees *)
        L : REAL ;			(* Length of the line *)

END_VAR

VAR_OUTPUT
	    x1 : REAL;			(* End x-coordinate *)
        y1 : REAL;			(* End y-coordinate *)
END_VAR
VAR
	        theta_rad : REAL;	(* Angle in radians *)
END_VAR

    theta_rad := theta * 3.14159265358979 / 180.0;  

	x1 := x0 + L * COS(theta_rad);
	y1 := y0 + L * SIN(theta_rad);

END_FUNCTION_BLOCK

// ---- FBs/FB_EnableAxes.TcPOU
FUNCTION_BLOCK FB_EnableAxes
VAR_INPUT
	bEnableAxes: BOOL := TRUE;
END_VAR
VAR_OUTPUT
	bAllAxesReady: BOOL := FALSE;
END_VAR
VAR_IN_OUT
	io_X: AXIS_REF;
	io_Y: AXIS_REF;
	io_Z: AXIS_REF;
	io_C: AXIS_REF;
	io_M1: AXIS_REF;
	io_M2: AXIS_REF;
	io_M3: AXIS_REF;
	io_M4 : AXIS_REF;
END_VAR
VAR
	fOverride: LREAL := 100.0;
	fbPowerX: MC_Power;
	fbPowerY: MC_Power;
	fbPowerZ: MC_Power;
	fbPowerC: MC_Power;	
	fbPowerM1: MC_Power;
	fbPowerM2: MC_Power;
	fbPowerM3: MC_Power;
	fbPowerM4 : MC_Power;

END_VAR

io_X.ReadStatus();
io_Y.ReadStatus();
io_Z.ReadStatus();
io_C.ReadStatus();

io_M1.ReadStatus();
io_M2.ReadStatus();
io_M3.ReadStatus();
io_M4.ReadStatus();


fbPowerX(
	Enable:=bEnableAxes, 
	Enable_Positive:=bEnableAxes, 
	Enable_Negative:=bEnableAxes, 
	Override:=fOverride, 
	BufferMode:= , 
	Axis:=io_X, 
	Status=> , 
	Busy=> , 
	Active=> , 
	Error=> , 
	ErrorID=> );
fbPowerY(
	Enable:=bEnableAxes, 
	Enable_Positive:=bEnableAxes, 
	Enable_Negative:=bEnableAxes, 
	Override:=fOverride, 
	BufferMode:= , 
	Axis:=io_Y, 
	Status=> , 
	Busy=> , 
	Active=> , 
	Error=> , 
	ErrorID=> );	
fbPowerZ(
	Enable:=bEnableAxes, 
	Enable_Positive:=bEnableAxes, 
	Enable_Negative:=bEnableAxes, 
	Override:=fOverride, 
	BufferMode:= , 
	Axis:=io_Z, 
	Status=> , 
	Busy=> , 
	Active=> , 
	Error=> , 
	ErrorID=> );
fbPowerC(
	Enable:=bEnableAxes, 
	Enable_Positive:=bEnableAxes, 
	Enable_Negative:=bEnableAxes, 
	Override:=fOverride, 
	BufferMode:= , 
	Axis:=io_C, 
	Status=> , 
	Busy=> , 
	Active=> , 
	Error=> , 
	ErrorID=> );
	
	
fbPowerM1(
	Enable:=bEnableAxes, 
	Enable_Positive:=bEnableAxes, 
	Enable_Negative:=bEnableAxes, 
	Override:=fOverride, 
	BufferMode:= , 
	Axis:=io_M1, 
	Status=> , 
	Busy=> , 
	Active=> , 
	Error=> , 
	ErrorID=> );	
fbPowerM2(
	Enable:=bEnableAxes, 
	Enable_Positive:=bEnableAxes, 
	Enable_Negative:=bEnableAxes, 
	Override:=fOverride, 
	BufferMode:= , 
	Axis:=io_M2, 
	Status=> , 
	Busy=> , 
	Active=> , 
	Error=> , 
	ErrorID=> );	
fbPowerM3(
	Enable:=bEnableAxes, 
	Enable_Positive:=bEnableAxes, 
	Enable_Negative:=bEnableAxes, 
	Override:=fOverride, 
	BufferMode:= , 
	Axis:=io_M3, 
	Status=> , 
	Busy=> , 
	Active=> , 
	Error=> , 
	ErrorID=> );	
fbPowerM4(
	Enable:=bEnableAxes, 
	Enable_Positive:=bEnableAxes, 
	Enable_Negative:=bEnableAxes, 
	Override:=fOverride, 
	BufferMode:= , 
	Axis:=io_M4, 
	Status=> , 
	Busy=> , 
	Active=> , 
	Error=> , 
	ErrorID=> );
	
bAllAxesReady	:= fbPowerX.Status AND fbPowerY.Status AND fbPowerZ.Status AND fbPowerC.Status AND  
	fbPowerM1.Status AND fbPowerM2.Status AND fbPowerM3.Status AND fbPowerM4.Status;

END_FUNCTION_BLOCK

// ---- FBs/FB_ResetCoordinateAxes.TcPOU
FUNCTION_BLOCK FB_ResetCoordinateAxes
VAR_INPUT
	resetAxes: BOOL := TRUE;
END_VAR
VAR_OUTPUT
	allAxesReset: BOOL := FALSE;
	error : BOOL;
	errorID : INT;
END_VAR
VAR_IN_OUT
	io_X: AXIS_REF;
	io_Y: AXIS_REF;
	io_Z: AXIS_REF;
	io_C: AXIS_REF;	
END_VAR
VAR
	fbResetX: MC_Reset;
	fbResetY: MC_Reset;
	fbResetZ: MC_Reset;
	fbResetC: MC_Reset;	
	fbResetM1: MC_Reset;
	fbResetM2: MC_Reset;
	fbResetM3: MC_Reset;
	fbResetM4: MC_Reset;
END_VAR


io_X.ReadStatus();
io_Y.ReadStatus();
io_Z.ReadStatus();
io_C.ReadStatus();


fbResetX(
	Execute:=resetAxes, 
	Axis:=io_X, 
	Done=> , 
	Busy=> , 
	Error=> , 
	ErrorID=> );
	
fbResetY(
	Execute:= fbResetX.Done, 
	Axis:=io_Y, 
	Done=> , 
	Busy=> , 
	Error=> , 
	ErrorID=> );
	
fbResetZ(
	Execute:= fbResetY.Done, 
	Axis:=io_Z, 
	Done=> , 
	Busy=> , 
	Error=> , 
	ErrorID=>  );
	
fbResetC(
	Execute:= fbResetZ.Done, 
	Axis:=io_C, 
	Done=> allAxesReset, 
	Busy=> , 
	Error=> , 
	ErrorID=>  );

END_FUNCTION_BLOCK
